_CFC_ (* Continuous Function Chart, elements in execution order *)
#0 RT_VKL_OLD_SEZ_LETO:R_TRIG(CLK: TRUE)
#1 MOVE(EN: #0.Q, SHU6_P2_UST_SEZ_LETO)
#2 SHU6_P2_UST_SEZ_LETO_OLD <= #1
#3 RT_VKL_OLD_SEZ_ZIMA:R_TRIG(CLK: TRUE)
#4 MOVE(EN: #3.Q, SHU6_P2_UST_SEZ_ZIMA)
#5 SHU6_P2_UST_SEZ_ZIMA_OLD <= #4
#6 <>(SHU6_P2_UST_SEZ_LETO, SHU6_P2_UST_SEZ_LETO_OLD)
#7 >(SHU6_P2_UST_SEZ_LETO, SHU6_P2_UST_SEZ_ZIMA_OLD)
#8 AND(#6, #7)
#9 MOVE(EN: #8, SHU6_P2_UST_SEZ_LETO)
#10 SHU6_P2_UST_SEZ_LETO_OLD <= #9
#11 AND(#6, NOT #7)
#12 MOVE(EN: #11, SHU6_P2_UST_SEZ_LETO_OLD)
#13 SHU6_P2_UST_SEZ_LETO <= #12
#14 <>(SHU6_P2_UST_SEZ_ZIMA, SHU6_P2_UST_SEZ_ZIMA_OLD)
#15 <(SHU6_P2_UST_SEZ_ZIMA, SHU6_P2_UST_SEZ_LETO_OLD)
#16 AND(#14, #15)
#17 MOVE(EN: #16, SHU6_P2_UST_SEZ_ZIMA)
#18 SHU6_P2_UST_SEZ_ZIMA_OLD <= #17
#19 AND(#14, NOT #15)
#20 MOVE(EN: #19, SHU6_P2_UST_SEZ_ZIMA_OLD)
#21 SHU6_P2_UST_SEZ_ZIMA <= #20
#22 RT_UE3_TE_UST_VKL_OLD:R_TRIG(CLK: TRUE)
#23 MOVE(EN: #22.Q, SHU6_P2_TE6_T_UST)
#24 SHU6_P2_TE6_T_UST_OLD <= #23
#25 <>(SHU6_P2_TE6_T_UST, SHU6_P2_TE6_T_UST_OLD)
#26 >(SHU6_P2_TE6_T_UST, SHU6_P2_UE1_T_UST_OLD)
#27 AND(#25, #26)
#28 MOVE(EN: #27, SHU6_P2_TE6_T_UST)
#29 SHU6_P2_TE6_T_UST_OLD <= #28
#30 AND(#25, NOT #26)
#31 MOVE(EN: #30, SHU6_P2_TE6_T_UST_OLD)
#32 SHU6_P2_TE6_T_UST <= #31
_END_CFC_
END_PROGRAM

(* POU Input/CI/MP2_1_OB, CFC *)
PROGRAM MP2_1_OB
VAR
	fb_M1_OBRbSM: ISTOK_GT;
	fb_M1b30: ISTOK_GT;
	fb_M1_OBRb45: ISTOK_GT;
	fb_M1_OBRm0_1: ISTOK_LT;
	fb_M_OBR: ISTOK_ANALOGVH;
	ofset: INT := 0;
	SR_DOST_M1: RS;
	dost_ton: TON;
END_VAR
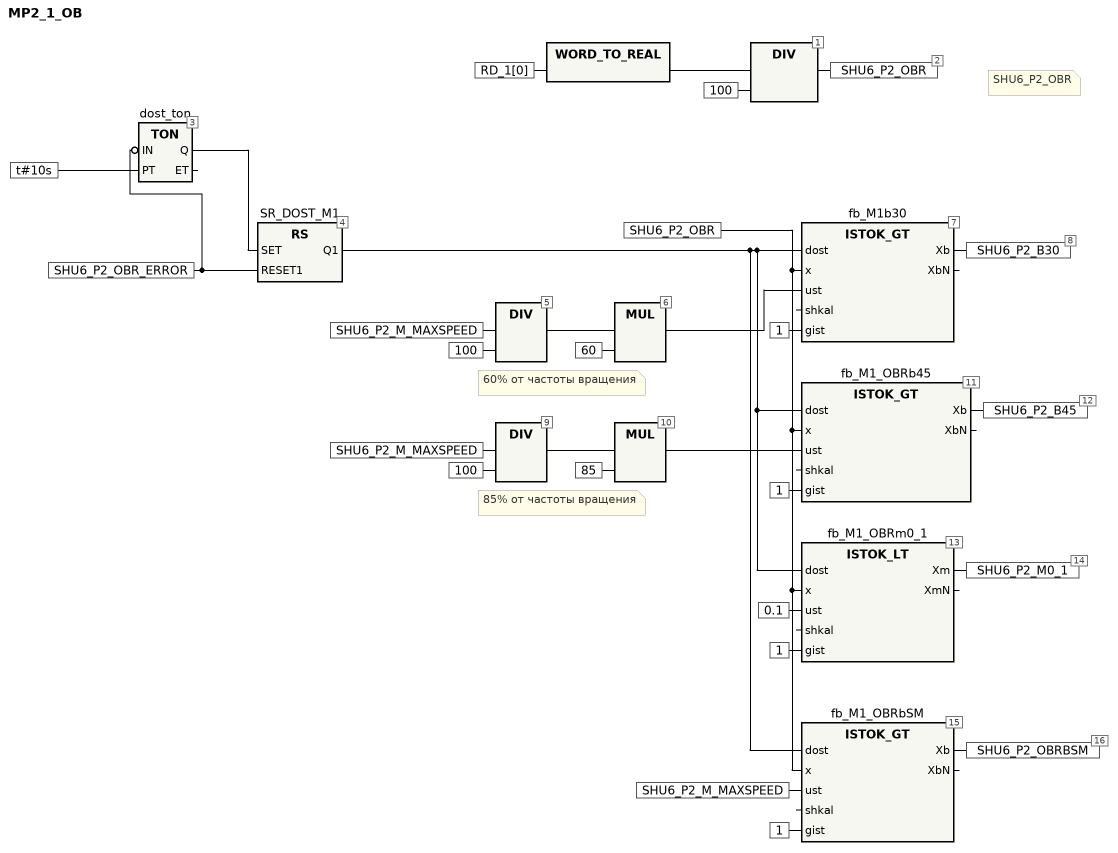
_CFC_ (* Continuous Function Chart, elements in execution order *)
(* SHU6_P2_OBR *)
(* 60% от частоты вращения *)
(* 85% от частоты вращения *)
#0 WORD_TO_REAL(RD_1[0])
#1 DIV(#0, 100)
#2 SHU6_P2_OBR <= #1
#3 dost_ton:TON(IN: NOT SHU6_P2_OBR_ERROR, PT: t#10s)
#4 SR_DOST_M1:RS(SET: #3.Q, RESET1: SHU6_P2_OBR_ERROR)
#5 DIV(SHU6_P2_M_MAXSPEED, 100)
#6 MUL(#5, 60)
#7 fb_M1b30:ISTOK_GT(dost: #4.Q1, x: SHU6_P2_OBR, ust: #6, shkal: -, gist: 1)
#8 SHU6_P2_B30 <= #7.Xb
#9 DIV(SHU6_P2_M_MAXSPEED, 100)
#10 MUL(#9, 85)
#11 fb_M1_OBRb45:ISTOK_GT(dost: #4.Q1, x: SHU6_P2_OBR, ust: #10, shkal: -, gist: 1)
#12 SHU6_P2_B45 <= #11.Xb
#13 fb_M1_OBRm0_1:ISTOK_LT(dost: #4.Q1, x: SHU6_P2_OBR, ust: 0.1, shkal: -, gist: 1)
#14 SHU6_P2_M0_1 <= #13.Xm
#15 fb_M1_OBRbSM:ISTOK_GT(dost: #4.Q1, x: SHU6_P2_OBR, ust: SHU6_P2_M_MAXSPEED, shkal: -, gist: 1)
#16 SHU6_P2_OBRBSM <= #15.Xb
_END_CFC_
(* the same logic as Structured Text *)
(* SHU6_P2_OBR *)
(* 60% от частоты вращения *)
(* 85% от частоты вращения *)
SHU6_P2_OBR := WORD_TO_REAL(RD_1[0]) / 100;
dost_ton(IN := NOT SHU6_P2_OBR_ERROR, PT := t#10s);
SR_DOST_M1(SET := dost_ton.Q, RESET1 := SHU6_P2_OBR_ERROR);
fb_M1b30(dost := SR_DOST_M1.Q1, x := SHU6_P2_OBR, ust := (SHU6_P2_M_MAXSPEED / 100) * 60, gist := 1);
SHU6_P2_B30 := fb_M1b30.Xb;
fb_M1_OBRb45(dost := SR_DOST_M1.Q1, x := SHU6_P2_OBR, ust := (SHU6_P2_M_MAXSPEED / 100) * 85, gist := 1);
SHU6_P2_B45 := fb_M1_OBRb45.Xb;
fb_M1_OBRm0_1(dost := SR_DOST_M1.Q1, x := SHU6_P2_OBR, ust := 0.1, gist := 1);
SHU6_P2_M0_1 := fb_M1_OBRm0_1.Xm;
fb_M1_OBRbSM(dost := SR_DOST_M1.Q1, x := SHU6_P2_OBR, ust := SHU6_P2_M_MAXSPEED, gist := 1);
SHU6_P2_OBRBSM := fb_M1_OBRbSM.Xb;
END_PROGRAM

(* POU Lib/ISTOK_GT, CFC *)
FUNCTION_BLOCK ISTOK_GT
VAR_INPUT
	dost: BOOL;
	x: REAL;
	ust: REAL;
	shkal: REAL;
	gist: REAL;
END_VAR
VAR_OUTPUT
	Xb: BOOL;
	XbN: BOOL;
END_VAR
VAR
	rs_gt: RS;
END_VAR
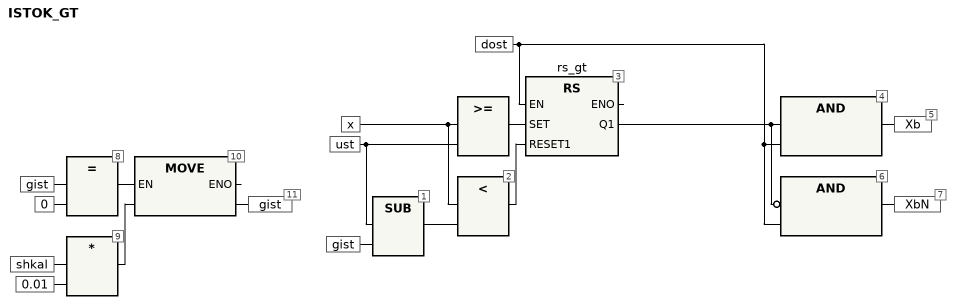
_CFC_ (* Continuous Function Chart, elements in execution order *)
#0 >=(x, ust)
#1 SUB(ust, gist)
#2 <(x, #1)
#3 rs_gt:RS(EN: dost, SET: #0, RESET1: #2)
#4 AND(#3.Q1, dost)
#5 Xb <= #4
#6 AND(NOT #3.Q1, dost)
#7 XbN <= #6
#8 =(gist, 0)
#9 *(shkal, 0.01)
#10 MOVE(EN: #8, #9)
#11 gist <= #10
_END_CFC_
END_FUNCTION_BLOCK

(* POU Lib/ISTOK_LT, CFC *)
FUNCTION_BLOCK ISTOK_LT
VAR_INPUT
	dost: BOOL;
	x: REAL;
	ust: REAL;
	shkal: REAL;
	gist: REAL;
END_VAR
VAR_OUTPUT
	Xm: BOOL;
	XmN: BOOL;
END_VAR
VAR
	rs_lt: RS;
END_VAR
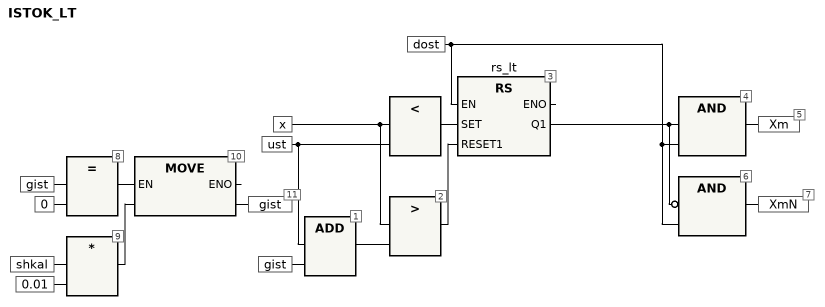
_CFC_ (* Continuous Function Chart, elements in execution order *)
#0 <(x, ust)
#1 ADD(ust, gist)
#2 >(x, #1)
#3 rs_lt:RS(EN: dost, SET: #0, RESET1: #2)
#4 AND(#3.Q1, dost)
#5 Xm <= #4
#6 AND(NOT #3.Q1, dost)
#7 XmN <= #6
#8 =(gist, 0)
#9 *(shkal, 0.01)
#10 MOVE(EN: #8, #9)
#11 gist <= #10
_END_CFC_
END_FUNCTION_BLOCK

(* POU Lib/ISTOK_ANALOGVH, CFC *)
FUNCTION_BLOCK ISTOK_ANALOGVH
VAR_INPUT
	enable: BOOL;
	rawValue: INT;
	reset: BOOL;
	enableLimitCtrl: BOOL;
	ctrlVoltage: BOOL;
	changeValueWithoutPower: BOOL := TRUE;

	highRange: REAL;
	lowRange: REAL;
	highLimit: REAL;
	lowLimit: REAL;
	filterTime: TIME;
	offset: REAL;

	delayEnable: TIME;
END_VAR
VAR_OUTPUT
	presentValue: REAL;
	byState: BYTE;
	byError: BYTE;

	reliability: BOOL;
	error: BOOL;
END_VAR
VAR
	fb_HVACAI: FB_HVACAnalogInput;

	bEnableLimitCtrl: BOOL := TRUE;

	iHighRange: INT := 32767;
	iLowRange: INT := 0;

	tFilterTime: TIME;
	rOffset: REAL := 0;

	delay: TON;

	a: BOOL;
	b: BOOL;
	c: INT;
	d: INT;
	delay_error: TON;
	SR_AI: SR;
	RS_AI: RS;

	I_GT: ISTOK_GT;
	I_LT: ISTOK_LT;
	TON_DOST: TON;
END_VAR
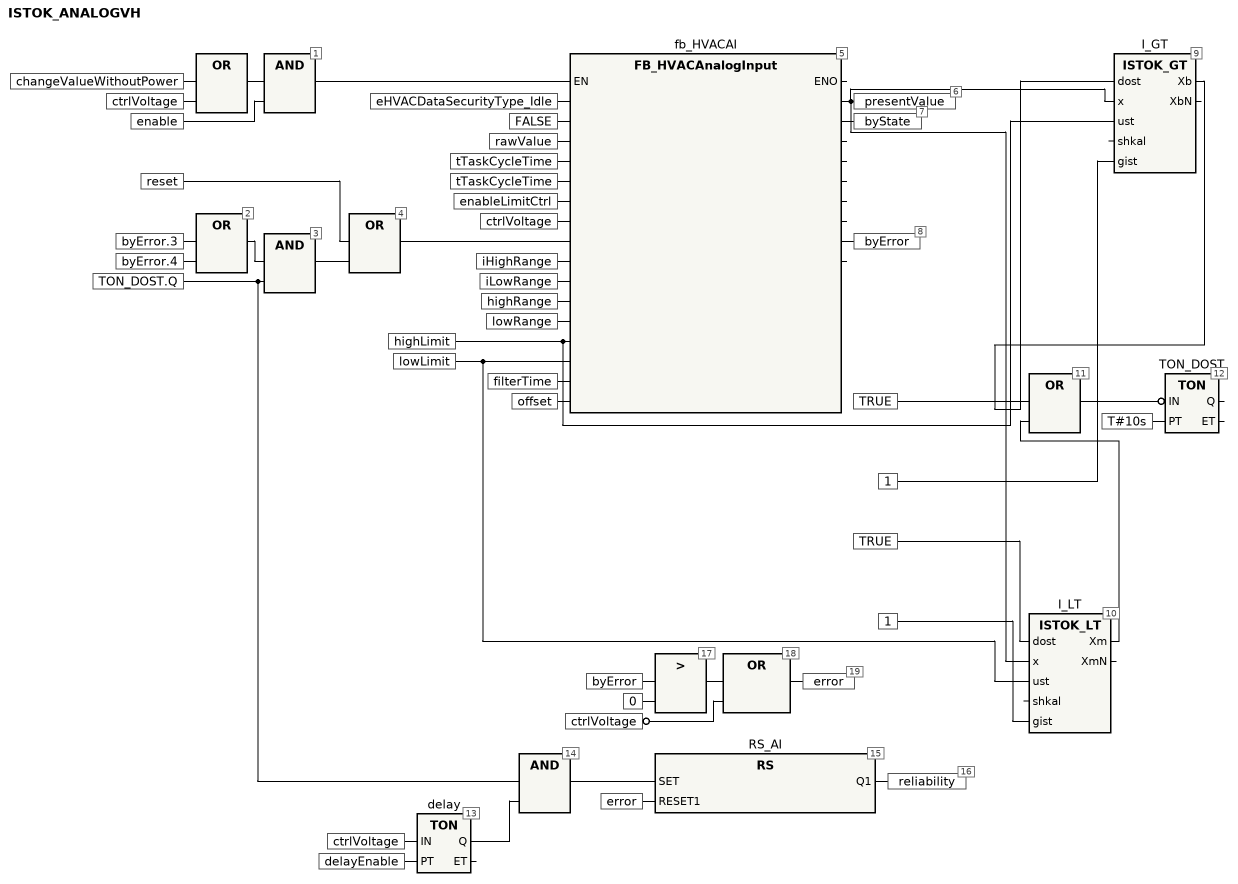
_CFC_ (* Continuous Function Chart, elements in execution order *)
#0 OR(changeValueWithoutPower, ctrlVoltage)
#1 AND(#0, enable)
#2 OR(byError.3, byError.4)
#3 AND(#2, TON_DOST.Q)
#4 OR(reset, #3)
#5 fb_HVACAI:FB_HVACAnalogInput(EN: #1, eHVACDataSecurityType_Idle, FALSE, rawValue, tTaskCycleTime, tTaskCycleTime, enableLimitCtrl, ctrlVoltage, #4, iHighRange, iLowRange, highRange, lowRange, highLimit, lowLimit, filterTime, offset)
#6 presentValue <= #5.out 1
#7 byState <= #5.out 2
#8 byError <= #5.out 8
#9 I_GT:ISTOK_GT(dost: TRUE, x: #5.out 1, ust: highLimit, shkal: -, gist: 1)
#10 I_LT:ISTOK_LT(dost: TRUE, x: #5.out 1, ust: lowLimit, shkal: -, gist: 1)
#11 OR(#9.Xb, #10.Xm)
#12 TON_DOST:TON(IN: NOT #11, PT: T#10s)
#13 delay:TON(IN: ctrlVoltage, PT: delayEnable)
#14 AND(TON_DOST.Q, #13.Q)
#15 RS_AI:RS(SET: #14, RESET1: error)
#16 reliability <= #15.Q1
#17 >(byError, 0)
#18 OR(#17, NOT ctrlVoltage)
#19 error <= #18
_END_CFC_
END_FUNCTION_BLOCK

(* POU Input/AI/TE1, CFC *)
PROGRAM TE1
VAR
	fb_TE1: ISTOK_ANALOGVH;
	ofset: REAL;
	fb_SHU6_P2_TE1_B_UST_MYAG_REG: ISTOK_GT;
	fb_SHU6_P2_TE1_B_UST_SEZ_LETO: ISTOK_GT;
	I_GT_TE: ISTOK_GT;
	I_LT_TE: ISTOK_LT;
	TON_DOST: TON;
END_VAR
VAR (* helpers for the ST form of the networks *)
	_t75 : REAL;
END_VAR
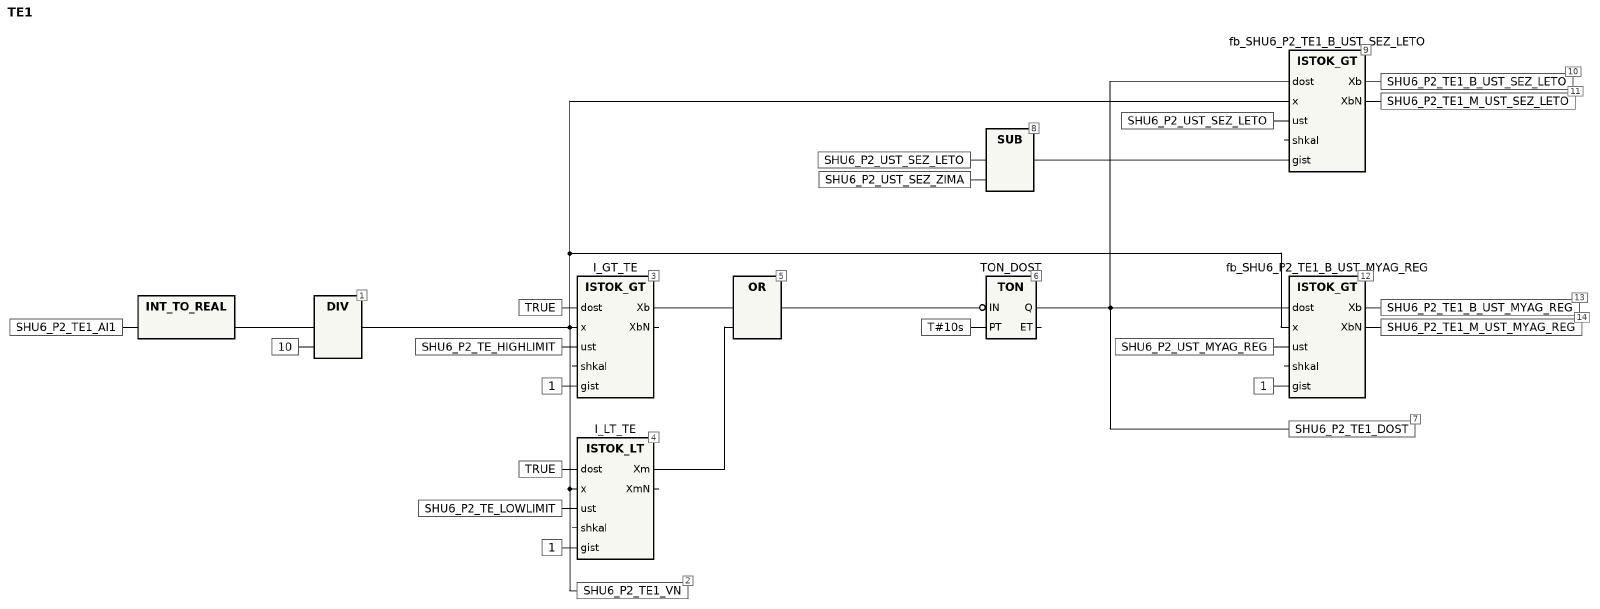
